{attribute 'qualified_only'}
VAR_GLOBAL
		EtherCAT_Master_EQxxxx : EtherCAT_Master_EQxxxx_26A48809;
END_VAR

(* stored: Version 1.2.0.0, ProductVersion 3.1.4024.9
   GVL GVL_iXlinker: Id {7d3bb3b1-94f9-49b9-b609-1719164548e6} *)
